// TIA Portal V15.1 export
// export: Created 2026-01-09T13:45:13.5597661Z, ExportSetting WithDefaults, WithReadOnly, DisplayName Totally Integrated Automation Portal, DisplayVersion V15.1 Update 8, DisplayName TIA Portal Openness, DisplayVersion V15.1 Update 8, DisplayName STEP 7 Professional, DisplayVersion V15.1 Update 8, DisplayName WinCC Advanced, DisplayVersion V15.1 Update 8
FUNCTION_BLOCK "11. LOGIC CAN"   // FB11, LAD
{ S7_Optimized_Access := 'TRUE' }
VERSION : 0.1
// stored: AutoNumber true, CodeModifiedDate 2025-08-27T17:14:05.4937984Z, CompileDate 2025-08-30T17:40:35.0335687Z, CreationDate 2024-10-12T12:36:08.0193576Z, DownloadWithoutReinit false, HandleErrorsWithinBlock false, InterfaceModifiedDate 2023-12-21T19:23:23.4270206Z, IsConsistent true, IsIECCheckEnabled false, IsKnowHowProtected false, IsRetainMemResEnabled false, IsWriteProtected false, LibraryConformanceStatus The object is library-conformant., MemoryReserve 100, ModifiedDate 2025-08-27T17:14:05.4937984Z, ParameterModified 2023-12-21T19:23:23.4270206Z, PLCSimAdvancedSupport false, SetENOAutomatically False, StructureModified 2023-12-21T19:23:23.4270206Z, UDAEnableTagReadback false
   VAR_INPUT
      LOGIC_1 : Real;
      LOGIC_2 : Real;
      LOGIC_3 : Real;
      "THC_1.1" : Bool;
      "THC_1.2" : Bool;
      "THC_2.1" : Bool;
      "THC_2.2" : Bool;
      "THC_3.1" : Bool;
      "THC_3.2" : Bool;
      "THC_4.1" : Bool;
      "THC_4.2" : Bool;
      "THC_5.1" : Bool;
      "THC_5.2" : Bool;
      "THC_6.1" : Bool;
      "THC_6.2" : Bool;
   END_VAR
   VAR_OUTPUT
      "OUT_LGOIC_1.1" : Bool;
      "OUT_LGOIC_1.2" : Bool;
      "OUT_LGOIC_2.1" : Bool;
      "OUT_LGOIC_2.2" : Bool;
      "OUT_LGOIC_3.1" : Bool;
      "OUT_LGOIC_3.2" : Bool;
      "OUT_LGOIC_4.1" : Bool;
      "OUT_LGOIC_4.2" : Bool;
      "OUT_LGOIC_5.1" : Bool;
      "OUT_LGOIC_5.2" : Bool;
      "OUT_LGOIC_6.1" : Bool;
      "OUT_LGOIC_6.2" : Bool;
   END_VAR
BEGIN

REGION Network 1: OUT1
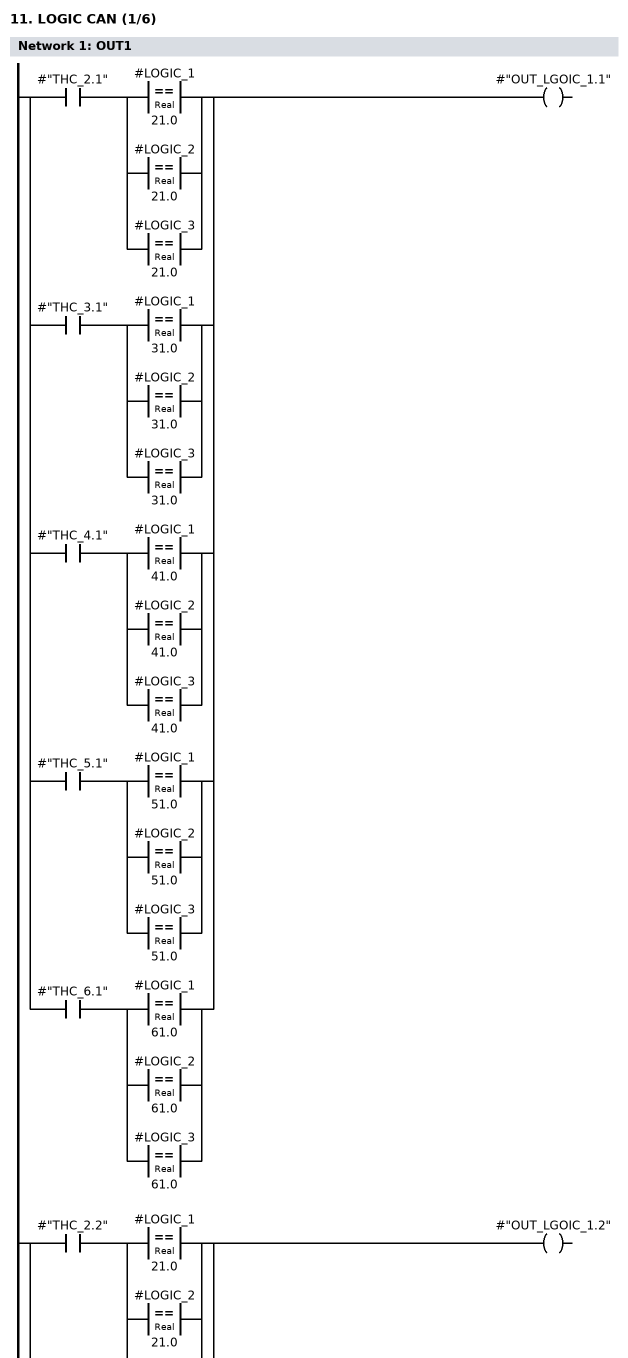
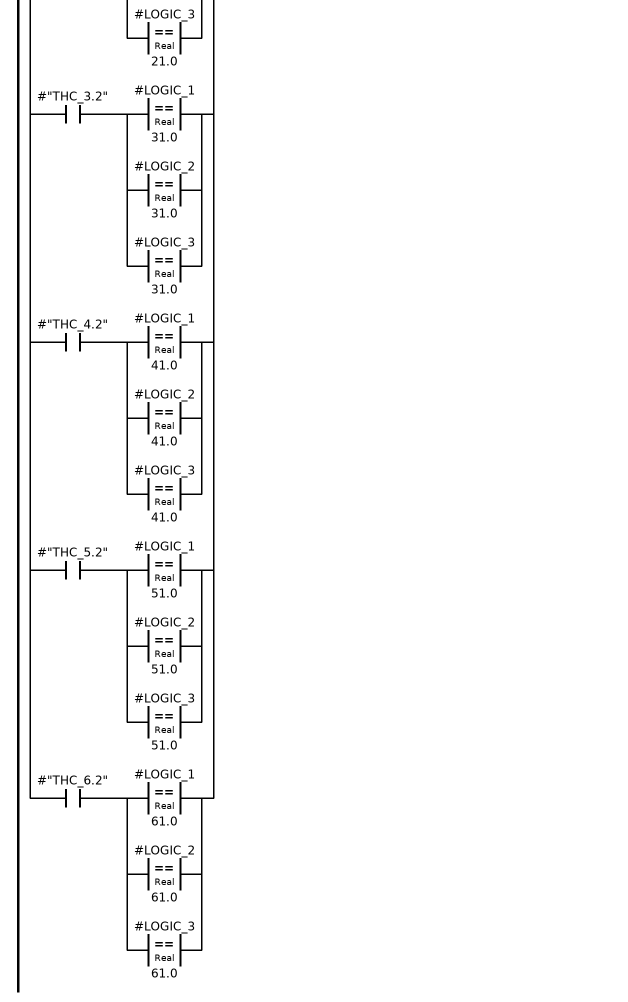
   RUNG wire#powerrail
      Contact( #"THC_2.1" )
      wire#w1
      { S7_Templates := "SrcType := Real" } EQ_Contact(in1 := #LOGIC_1, in2 := 21.0)
      wire#w2
      Coil( #"OUT_LGOIC_1.1" )
   END_RUNG
   RUNG wire#w1
      { S7_Templates := "SrcType := Real" } EQ_Contact(in1 := #LOGIC_2, in2 := 21.0)
   END_RUNG wire#w2
   RUNG wire#w1
      { S7_Templates := "SrcType := Real" } EQ_Contact(in1 := #LOGIC_3, in2 := 21.0)
   END_RUNG wire#w2
   RUNG wire#powerrail
      Contact( #"THC_3.1" )
      wire#w3
      { S7_Templates := "SrcType := Real" } EQ_Contact(in1 := #LOGIC_1, in2 := 31.0)
   END_RUNG wire#w2
   RUNG wire#w3
      { S7_Templates := "SrcType := Real" } EQ_Contact(in1 := #LOGIC_2, in2 := 31.0)
   END_RUNG wire#w2
   RUNG wire#w3
      { S7_Templates := "SrcType := Real" } EQ_Contact(in1 := #LOGIC_3, in2 := 31.0)
   END_RUNG wire#w2
   RUNG wire#powerrail
      Contact( #"THC_4.1" )
      wire#w4
      { S7_Templates := "SrcType := Real" } EQ_Contact(in1 := #LOGIC_1, in2 := 41.0)
   END_RUNG wire#w2
   RUNG wire#w4
      { S7_Templates := "SrcType := Real" } EQ_Contact(in1 := #LOGIC_2, in2 := 41.0)
   END_RUNG wire#w2
   RUNG wire#w4
      { S7_Templates := "SrcType := Real" } EQ_Contact(in1 := #LOGIC_3, in2 := 41.0)
   END_RUNG wire#w2
   RUNG wire#powerrail
      Contact( #"THC_5.1" )
      wire#w5
      { S7_Templates := "SrcType := Real" } EQ_Contact(in1 := #LOGIC_1, in2 := 51.0)
   END_RUNG wire#w2
   RUNG wire#w5
      { S7_Templates := "SrcType := Real" } EQ_Contact(in1 := #LOGIC_2, in2 := 51.0)
   END_RUNG wire#w2
   RUNG wire#w5
      { S7_Templates := "SrcType := Real" } EQ_Contact(in1 := #LOGIC_3, in2 := 51.0)
   END_RUNG wire#w2
   RUNG wire#powerrail
      Contact( #"THC_6.1" )
      wire#w6
      { S7_Templates := "SrcType := Real" } EQ_Contact(in1 := #LOGIC_1, in2 := 61.0)
   END_RUNG wire#w2
   RUNG wire#w6
      { S7_Templates := "SrcType := Real" } EQ_Contact(in1 := #LOGIC_2, in2 := 61.0)
   END_RUNG wire#w2
   RUNG wire#w6
      { S7_Templates := "SrcType := Real" } EQ_Contact(in1 := #LOGIC_3, in2 := 61.0)
   END_RUNG wire#w2
   RUNG wire#powerrail
      Contact( #"THC_2.2" )
      wire#w7
      { S7_Templates := "SrcType := Real" } EQ_Contact(in1 := #LOGIC_1, in2 := 21.0)
      wire#w8
      Coil( #"OUT_LGOIC_1.2" )
   END_RUNG
   RUNG wire#w7
      { S7_Templates := "SrcType := Real" } EQ_Contact(in1 := #LOGIC_2, in2 := 21.0)
   END_RUNG wire#w8
   RUNG wire#w7
      { S7_Templates := "SrcType := Real" } EQ_Contact(in1 := #LOGIC_3, in2 := 21.0)
   END_RUNG wire#w8
   RUNG wire#powerrail
      Contact( #"THC_3.2" )
      wire#w9
      { S7_Templates := "SrcType := Real" } EQ_Contact(in1 := #LOGIC_1, in2 := 31.0)
   END_RUNG wire#w8
   RUNG wire#w9
      { S7_Templates := "SrcType := Real" } EQ_Contact(in1 := #LOGIC_2, in2 := 31.0)
   END_RUNG wire#w8
   RUNG wire#w9
      { S7_Templates := "SrcType := Real" } EQ_Contact(in1 := #LOGIC_3, in2 := 31.0)
   END_RUNG wire#w8
   RUNG wire#powerrail
      Contact( #"THC_4.2" )
      wire#w10
      { S7_Templates := "SrcType := Real" } EQ_Contact(in1 := #LOGIC_1, in2 := 41.0)
   END_RUNG wire#w8
   RUNG wire#w10
      { S7_Templates := "SrcType := Real" } EQ_Contact(in1 := #LOGIC_2, in2 := 41.0)
   END_RUNG wire#w8
   RUNG wire#w10
      { S7_Templates := "SrcType := Real" } EQ_Contact(in1 := #LOGIC_3, in2 := 41.0)
   END_RUNG wire#w8
   RUNG wire#powerrail
      Contact( #"THC_5.2" )
      wire#w11
      { S7_Templates := "SrcType := Real" } EQ_Contact(in1 := #LOGIC_1, in2 := 51.0)
   END_RUNG wire#w8
   RUNG wire#w11
      { S7_Templates := "SrcType := Real" } EQ_Contact(in1 := #LOGIC_2, in2 := 51.0)
   END_RUNG wire#w8
   RUNG wire#w11
      { S7_Templates := "SrcType := Real" } EQ_Contact(in1 := #LOGIC_3, in2 := 51.0)
   END_RUNG wire#w8
   RUNG wire#powerrail
      Contact( #"THC_6.2" )
      wire#w12
      { S7_Templates := "SrcType := Real" } EQ_Contact(in1 := #LOGIC_1, in2 := 61.0)
   END_RUNG wire#w8
   RUNG wire#w12
      { S7_Templates := "SrcType := Real" } EQ_Contact(in1 := #LOGIC_2, in2 := 61.0)
   END_RUNG wire#w8
   RUNG wire#w12
      { S7_Templates := "SrcType := Real" } EQ_Contact(in1 := #LOGIC_3, in2 := 61.0)
   END_RUNG wire#w8
   // the same network as SCL:
   #"OUT_LGOIC_1.1" := (#"THC_2.1" AND ((#LOGIC_1 = 21.0) OR (#LOGIC_2 = 21.0) OR (#LOGIC_3 = 21.0))) OR (#"THC_3.1" AND ((#LOGIC_1 = 31.0) OR (#LOGIC_2 = 31.0) OR (#LOGIC_3 = 31.0))) OR (#"THC_4.1" AND ((#LOGIC_1 = 41.0) OR (#LOGIC_2 = 41.0) OR (#LOGIC_3 = 41.0))) OR (#"THC_5.1" AND ((#LOGIC_1 = 51.0) OR (#LOGIC_2 = 51.0) OR (#LOGIC_3 = 51.0))) OR (#"THC_6.1" AND ((#LOGIC_1 = 61.0) OR (#LOGIC_2 = 61.0) OR (#LOGIC_3 = 61.0)));
   #"OUT_LGOIC_1.2" := (#"THC_2.2" AND ((#LOGIC_1 = 21.0) OR (#LOGIC_2 = 21.0) OR (#LOGIC_3 = 21.0))) OR (#"THC_3.2" AND ((#LOGIC_1 = 31.0) OR (#LOGIC_2 = 31.0) OR (#LOGIC_3 = 31.0))) OR (#"THC_4.2" AND ((#LOGIC_1 = 41.0) OR (#LOGIC_2 = 41.0) OR (#LOGIC_3 = 41.0))) OR (#"THC_5.2" AND ((#LOGIC_1 = 51.0) OR (#LOGIC_2 = 51.0) OR (#LOGIC_3 = 51.0))) OR (#"THC_6.2" AND ((#LOGIC_1 = 61.0) OR (#LOGIC_2 = 61.0) OR (#LOGIC_3 = 61.0)));
END_REGION

REGION Network 2: OUT2
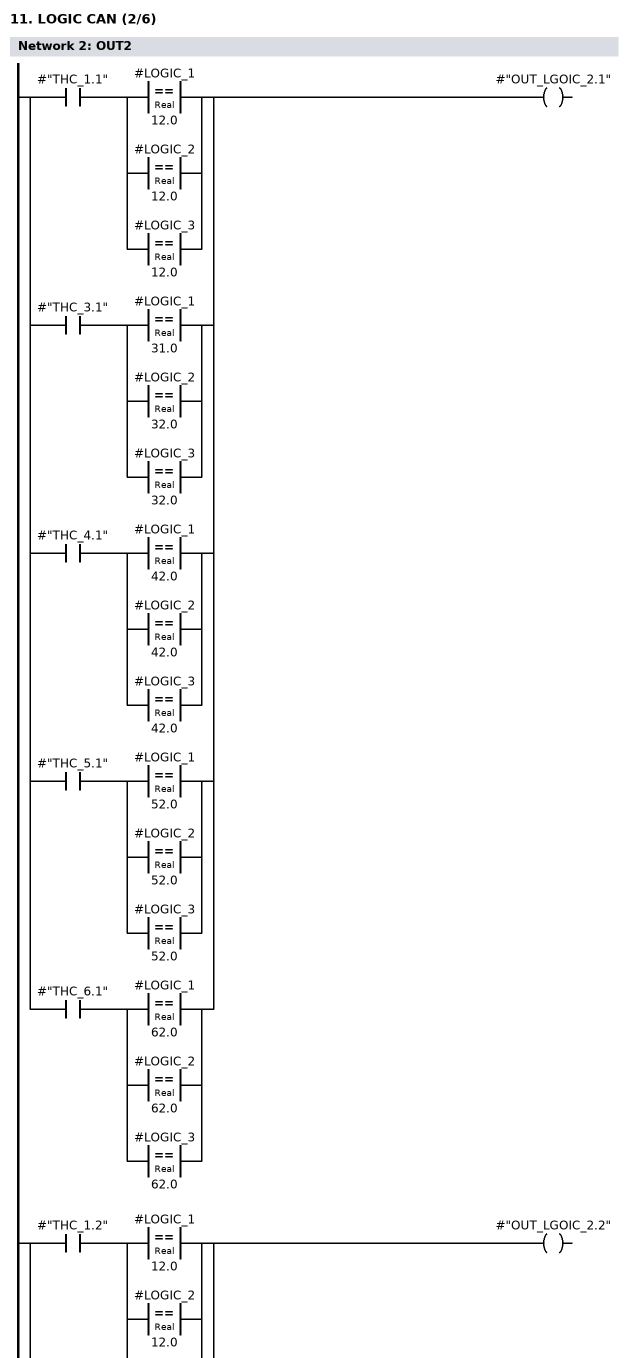
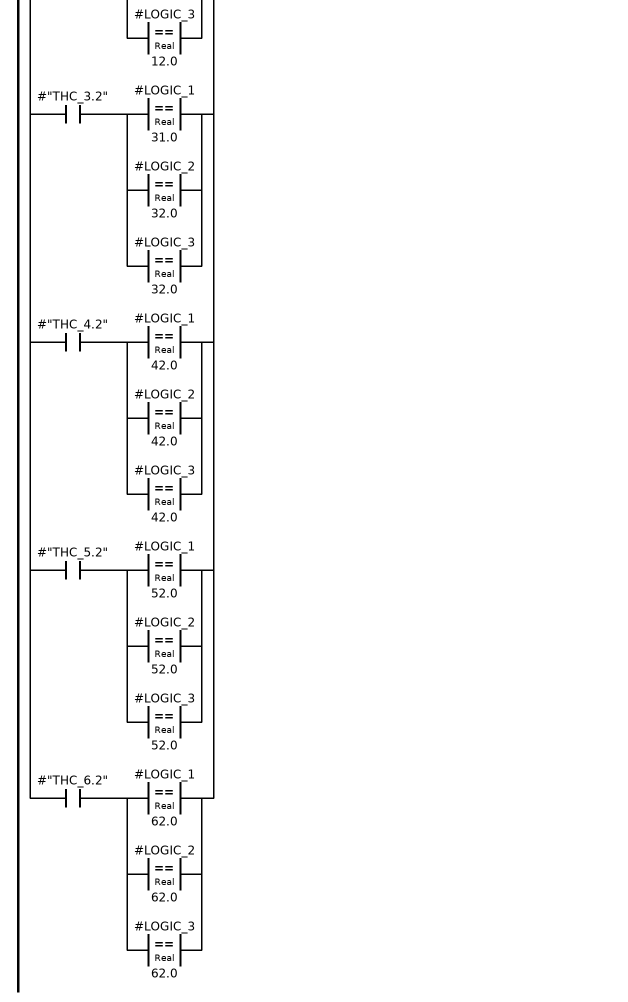
   RUNG wire#powerrail
      Contact( #"THC_1.1" )
      wire#w1
      { S7_Templates := "SrcType := Real" } EQ_Contact(in1 := #LOGIC_1, in2 := 12.0)
      wire#w2
      Coil( #"OUT_LGOIC_2.1" )
   END_RUNG
   RUNG wire#w1
      { S7_Templates := "SrcType := Real" } EQ_Contact(in1 := #LOGIC_2, in2 := 12.0)
   END_RUNG wire#w2
   RUNG wire#w1
      { S7_Templates := "SrcType := Real" } EQ_Contact(in1 := #LOGIC_3, in2 := 12.0)
   END_RUNG wire#w2
   RUNG wire#powerrail
      Contact( #"THC_3.1" )
      wire#w3
      { S7_Templates := "SrcType := Real" } EQ_Contact(in1 := #LOGIC_1, in2 := 31.0)
   END_RUNG wire#w2
   RUNG wire#w3
      { S7_Templates := "SrcType := Real" } EQ_Contact(in1 := #LOGIC_2, in2 := 32.0)
   END_RUNG wire#w2
   RUNG wire#w3
      { S7_Templates := "SrcType := Real" } EQ_Contact(in1 := #LOGIC_3, in2 := 32.0)
   END_RUNG wire#w2
   RUNG wire#powerrail
      Contact( #"THC_4.1" )
      wire#w4
      { S7_Templates := "SrcType := Real" } EQ_Contact(in1 := #LOGIC_1, in2 := 42.0)
   END_RUNG wire#w2
   RUNG wire#w4
      { S7_Templates := "SrcType := Real" } EQ_Contact(in1 := #LOGIC_2, in2 := 42.0)
   END_RUNG wire#w2
   RUNG wire#w4
      { S7_Templates := "SrcType := Real" } EQ_Contact(in1 := #LOGIC_3, in2 := 42.0)
   END_RUNG wire#w2
   RUNG wire#powerrail
      Contact( #"THC_5.1" )
      wire#w5
      { S7_Templates := "SrcType := Real" } EQ_Contact(in1 := #LOGIC_1, in2 := 52.0)
   END_RUNG wire#w2
   RUNG wire#w5
      { S7_Templates := "SrcType := Real" } EQ_Contact(in1 := #LOGIC_2, in2 := 52.0)
   END_RUNG wire#w2
   RUNG wire#w5
      { S7_Templates := "SrcType := Real" } EQ_Contact(in1 := #LOGIC_3, in2 := 52.0)
   END_RUNG wire#w2
   RUNG wire#powerrail
      Contact( #"THC_6.1" )
      wire#w6
      { S7_Templates := "SrcType := Real" } EQ_Contact(in1 := #LOGIC_1, in2 := 62.0)
   END_RUNG wire#w2
   RUNG wire#w6
      { S7_Templates := "SrcType := Real" } EQ_Contact(in1 := #LOGIC_2, in2 := 62.0)
   END_RUNG wire#w2
   RUNG wire#w6
      { S7_Templates := "SrcType := Real" } EQ_Contact(in1 := #LOGIC_3, in2 := 62.0)
   END_RUNG wire#w2
   RUNG wire#powerrail
      Contact( #"THC_1.2" )
      wire#w7
      { S7_Templates := "SrcType := Real" } EQ_Contact(in1 := #LOGIC_1, in2 := 12.0)
      wire#w8
      Coil( #"OUT_LGOIC_2.2" )
   END_RUNG
   RUNG wire#w7
      { S7_Templates := "SrcType := Real" } EQ_Contact(in1 := #LOGIC_2, in2 := 12.0)
   END_RUNG wire#w8
   RUNG wire#w7
      { S7_Templates := "SrcType := Real" } EQ_Contact(in1 := #LOGIC_3, in2 := 12.0)
   END_RUNG wire#w8
   RUNG wire#powerrail
      Contact( #"THC_3.2" )
      wire#w9
      { S7_Templates := "SrcType := Real" } EQ_Contact(in1 := #LOGIC_1, in2 := 31.0)
   END_RUNG wire#w8
   RUNG wire#w9
      { S7_Templates := "SrcType := Real" } EQ_Contact(in1 := #LOGIC_2, in2 := 32.0)
   END_RUNG wire#w8
   RUNG wire#w9
      { S7_Templates := "SrcType := Real" } EQ_Contact(in1 := #LOGIC_3, in2 := 32.0)
   END_RUNG wire#w8
   RUNG wire#powerrail
      Contact( #"THC_4.2" )
      wire#w10
      { S7_Templates := "SrcType := Real" } EQ_Contact(in1 := #LOGIC_1, in2 := 42.0)
   END_RUNG wire#w8
   RUNG wire#w10
      { S7_Templates := "SrcType := Real" } EQ_Contact(in1 := #LOGIC_2, in2 := 42.0)
   END_RUNG wire#w8
   RUNG wire#w10
      { S7_Templates := "SrcType := Real" } EQ_Contact(in1 := #LOGIC_3, in2 := 42.0)
   END_RUNG wire#w8
   RUNG wire#powerrail
      Contact( #"THC_5.2" )
      wire#w11
      { S7_Templates := "SrcType := Real" } EQ_Contact(in1 := #LOGIC_1, in2 := 52.0)
   END_RUNG wire#w8
   RUNG wire#w11
      { S7_Templates := "SrcType := Real" } EQ_Contact(in1 := #LOGIC_2, in2 := 52.0)
   END_RUNG wire#w8
   RUNG wire#w11
      { S7_Templates := "SrcType := Real" } EQ_Contact(in1 := #LOGIC_3, in2 := 52.0)
   END_RUNG wire#w8
   RUNG wire#powerrail
      Contact( #"THC_6.2" )
      wire#w12
      { S7_Templates := "SrcType := Real" } EQ_Contact(in1 := #LOGIC_1, in2 := 62.0)
   END_RUNG wire#w8
   RUNG wire#w12
      { S7_Templates := "SrcType := Real" } EQ_Contact(in1 := #LOGIC_2, in2 := 62.0)
   END_RUNG wire#w8
   RUNG wire#w12
      { S7_Templates := "SrcType := Real" } EQ_Contact(in1 := #LOGIC_3, in2 := 62.0)
   END_RUNG wire#w8
   // the same network as SCL:
   #"OUT_LGOIC_2.1" := (#"THC_1.1" AND ((#LOGIC_1 = 12.0) OR (#LOGIC_2 = 12.0) OR (#LOGIC_3 = 12.0))) OR (#"THC_3.1" AND ((#LOGIC_1 = 31.0) OR (#LOGIC_2 = 32.0) OR (#LOGIC_3 = 32.0))) OR (#"THC_4.1" AND ((#LOGIC_1 = 42.0) OR (#LOGIC_2 = 42.0) OR (#LOGIC_3 = 42.0))) OR (#"THC_5.1" AND ((#LOGIC_1 = 52.0) OR (#LOGIC_2 = 52.0) OR (#LOGIC_3 = 52.0))) OR (#"THC_6.1" AND ((#LOGIC_1 = 62.0) OR (#LOGIC_2 = 62.0) OR (#LOGIC_3 = 62.0)));
   #"OUT_LGOIC_2.2" := (#"THC_1.2" AND ((#LOGIC_1 = 12.0) OR (#LOGIC_2 = 12.0) OR (#LOGIC_3 = 12.0))) OR (#"THC_3.2" AND ((#LOGIC_1 = 31.0) OR (#LOGIC_2 = 32.0) OR (#LOGIC_3 = 32.0))) OR (#"THC_4.2" AND ((#LOGIC_1 = 42.0) OR (#LOGIC_2 = 42.0) OR (#LOGIC_3 = 42.0))) OR (#"THC_5.2" AND ((#LOGIC_1 = 52.0) OR (#LOGIC_2 = 52.0) OR (#LOGIC_3 = 52.0))) OR (#"THC_6.2" AND ((#LOGIC_1 = 62.0) OR (#LOGIC_2 = 62.0) OR (#LOGIC_3 = 62.0)));
END_REGION

REGION Network 3: OUT3
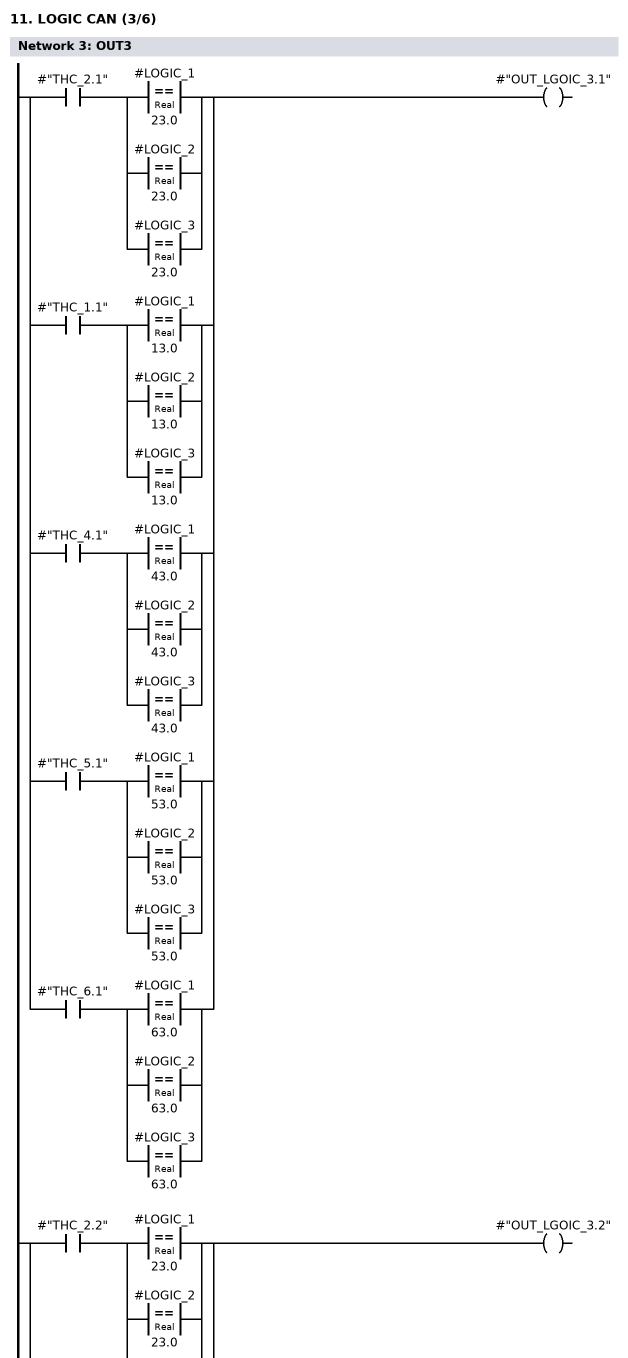
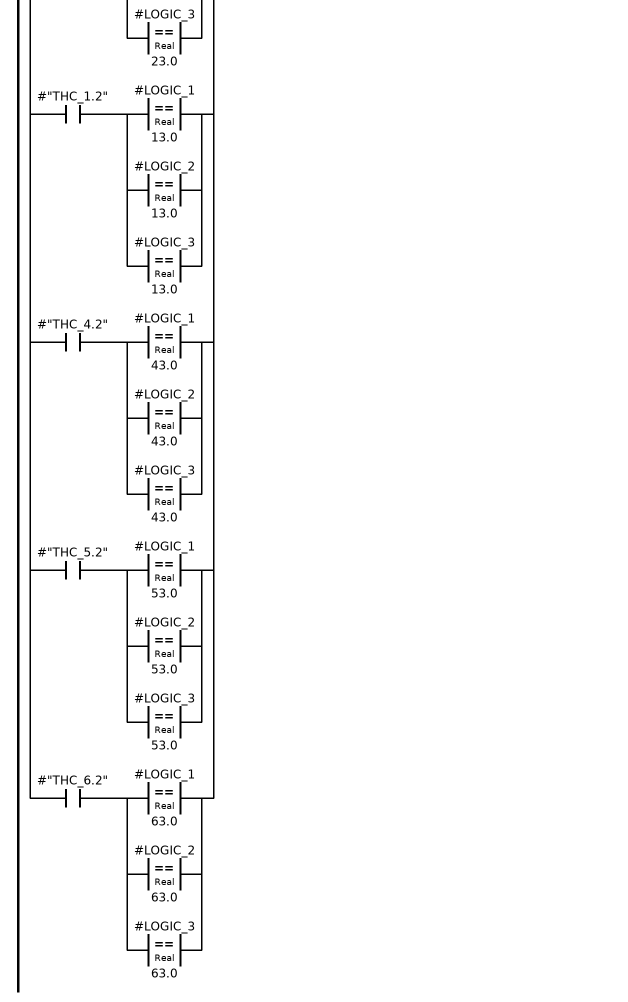
   RUNG wire#powerrail
      Contact( #"THC_2.1" )
      wire#w1
      { S7_Templates := "SrcType := Real" } EQ_Contact(in1 := #LOGIC_1, in2 := 23.0)
      wire#w2
      Coil( #"OUT_LGOIC_3.1" )
   END_RUNG
   RUNG wire#w1
      { S7_Templates := "SrcType := Real" } EQ_Contact(in1 := #LOGIC_2, in2 := 23.0)
   END_RUNG wire#w2
   RUNG wire#w1
      { S7_Templates := "SrcType := Real" } EQ_Contact(in1 := #LOGIC_3, in2 := 23.0)
   END_RUNG wire#w2
   RUNG wire#powerrail
      Contact( #"THC_1.1" )
      wire#w3
      { S7_Templates := "SrcType := Real" } EQ_Contact(in1 := #LOGIC_1, in2 := 13.0)
   END_RUNG wire#w2
   RUNG wire#w3
      { S7_Templates := "SrcType := Real" } EQ_Contact(in1 := #LOGIC_2, in2 := 13.0)
   END_RUNG wire#w2
   RUNG wire#w3
      { S7_Templates := "SrcType := Real" } EQ_Contact(in1 := #LOGIC_3, in2 := 13.0)
   END_RUNG wire#w2
   RUNG wire#powerrail
      Contact( #"THC_4.1" )
      wire#w4
      { S7_Templates := "SrcType := Real" } EQ_Contact(in1 := #LOGIC_1, in2 := 43.0)
   END_RUNG wire#w2
   RUNG wire#w4
      { S7_Templates := "SrcType := Real" } EQ_Contact(in1 := #LOGIC_2, in2 := 43.0)
   END_RUNG wire#w2
   RUNG wire#w4
      { S7_Templates := "SrcType := Real" } EQ_Contact(in1 := #LOGIC_3, in2 := 43.0)
   END_RUNG wire#w2
   RUNG wire#powerrail
      Contact( #"THC_5.1" )
      wire#w5
      { S7_Templates := "SrcType := Real" } EQ_Contact(in1 := #LOGIC_1, in2 := 53.0)
   END_RUNG wire#w2
   RUNG wire#w5
      { S7_Templates := "SrcType := Real" } EQ_Contact(in1 := #LOGIC_2, in2 := 53.0)
   END_RUNG wire#w2
   RUNG wire#w5
      { S7_Templates := "SrcType := Real" } EQ_Contact(in1 := #LOGIC_3, in2 := 53.0)
   END_RUNG wire#w2
   RUNG wire#powerrail
      Contact( #"THC_6.1" )
      wire#w6
      { S7_Templates := "SrcType := Real" } EQ_Contact(in1 := #LOGIC_1, in2 := 63.0)
   END_RUNG wire#w2
   RUNG wire#w6
      { S7_Templates := "SrcType := Real" } EQ_Contact(in1 := #LOGIC_2, in2 := 63.0)
   END_RUNG wire#w2
   RUNG wire#w6
      { S7_Templates := "SrcType := Real" } EQ_Contact(in1 := #LOGIC_3, in2 := 63.0)
   END_RUNG wire#w2
   RUNG wire#powerrail
      Contact( #"THC_2.2" )
      wire#w7
      { S7_Templates := "SrcType := Real" } EQ_Contact(in1 := #LOGIC_1, in2 := 23.0)
      wire#w8
      Coil( #"OUT_LGOIC_3.2" )
   END_RUNG
   RUNG wire#w7
      { S7_Templates := "SrcType := Real" } EQ_Contact(in1 := #LOGIC_2, in2 := 23.0)
   END_RUNG wire#w8
   RUNG wire#w7
      { S7_Templates := "SrcType := Real" } EQ_Contact(in1 := #LOGIC_3, in2 := 23.0)
   END_RUNG wire#w8
   RUNG wire#powerrail
      Contact( #"THC_1.2" )
      wire#w9
      { S7_Templates := "SrcType := Real" } EQ_Contact(in1 := #LOGIC_1, in2 := 13.0)
   END_RUNG wire#w8
   RUNG wire#w9
      { S7_Templates := "SrcType := Real" } EQ_Contact(in1 := #LOGIC_2, in2 := 13.0)
   END_RUNG wire#w8
   RUNG wire#w9
      { S7_Templates := "SrcType := Real" } EQ_Contact(in1 := #LOGIC_3, in2 := 13.0)
   END_RUNG wire#w8
   RUNG wire#powerrail
      Contact( #"THC_4.2" )
      wire#w10
      { S7_Templates := "SrcType := Real" } EQ_Contact(in1 := #LOGIC_1, in2 := 43.0)
   END_RUNG wire#w8
   RUNG wire#w10
      { S7_Templates := "SrcType := Real" } EQ_Contact(in1 := #LOGIC_2, in2 := 43.0)
   END_RUNG wire#w8
   RUNG wire#w10
      { S7_Templates := "SrcType := Real" } EQ_Contact(in1 := #LOGIC_3, in2 := 43.0)
   END_RUNG wire#w8
   RUNG wire#powerrail
      Contact( #"THC_5.2" )
      wire#w11
      { S7_Templates := "SrcType := Real" } EQ_Contact(in1 := #LOGIC_1, in2 := 53.0)
   END_RUNG wire#w8
   RUNG wire#w11
      { S7_Templates := "SrcType := Real" } EQ_Contact(in1 := #LOGIC_2, in2 := 53.0)
   END_RUNG wire#w8
   RUNG wire#w11
      { S7_Templates := "SrcType := Real" } EQ_Contact(in1 := #LOGIC_3, in2 := 53.0)
   END_RUNG wire#w8
   RUNG wire#powerrail
      Contact( #"THC_6.2" )
      wire#w12
      { S7_Templates := "SrcType := Real" } EQ_Contact(in1 := #LOGIC_1, in2 := 63.0)
   END_RUNG wire#w8
   RUNG wire#w12
      { S7_Templates := "SrcType := Real" } EQ_Contact(in1 := #LOGIC_2, in2 := 63.0)
   END_RUNG wire#w8
   RUNG wire#w12
      { S7_Templates := "SrcType := Real" } EQ_Contact(in1 := #LOGIC_3, in2 := 63.0)
   END_RUNG wire#w8
   // the same network as SCL:
   #"OUT_LGOIC_3.1" := (#"THC_2.1" AND ((#LOGIC_1 = 23.0) OR (#LOGIC_2 = 23.0) OR (#LOGIC_3 = 23.0))) OR (#"THC_1.1" AND ((#LOGIC_1 = 13.0) OR (#LOGIC_2 = 13.0) OR (#LOGIC_3 = 13.0))) OR (#"THC_4.1" AND ((#LOGIC_1 = 43.0) OR (#LOGIC_2 = 43.0) OR (#LOGIC_3 = 43.0))) OR (#"THC_5.1" AND ((#LOGIC_1 = 53.0) OR (#LOGIC_2 = 53.0) OR (#LOGIC_3 = 53.0))) OR (#"THC_6.1" AND ((#LOGIC_1 = 63.0) OR (#LOGIC_2 = 63.0) OR (#LOGIC_3 = 63.0)));
   #"OUT_LGOIC_3.2" := (#"THC_2.2" AND ((#LOGIC_1 = 23.0) OR (#LOGIC_2 = 23.0) OR (#LOGIC_3 = 23.0))) OR (#"THC_1.2" AND ((#LOGIC_1 = 13.0) OR (#LOGIC_2 = 13.0) OR (#LOGIC_3 = 13.0))) OR (#"THC_4.2" AND ((#LOGIC_1 = 43.0) OR (#LOGIC_2 = 43.0) OR (#LOGIC_3 = 43.0))) OR (#"THC_5.2" AND ((#LOGIC_1 = 53.0) OR (#LOGIC_2 = 53.0) OR (#LOGIC_3 = 53.0))) OR (#"THC_6.2" AND ((#LOGIC_1 = 63.0) OR (#LOGIC_2 = 63.0) OR (#LOGIC_3 = 63.0)));
END_REGION

REGION Network 4: OUT4
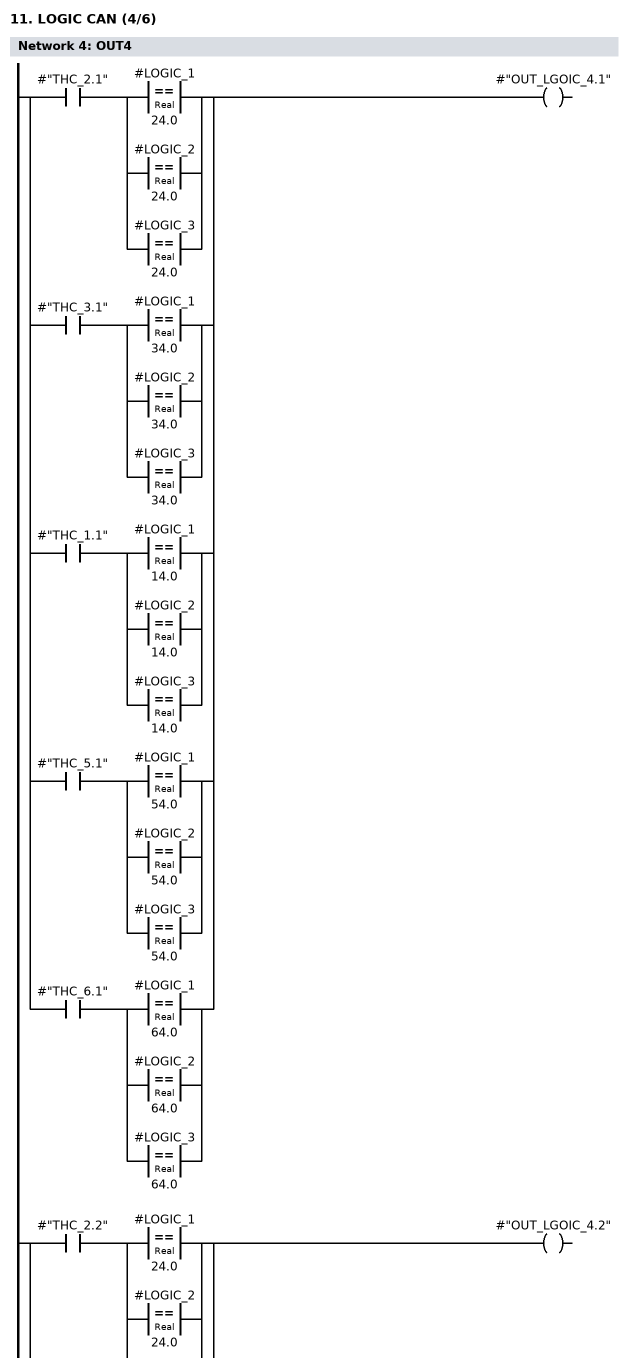
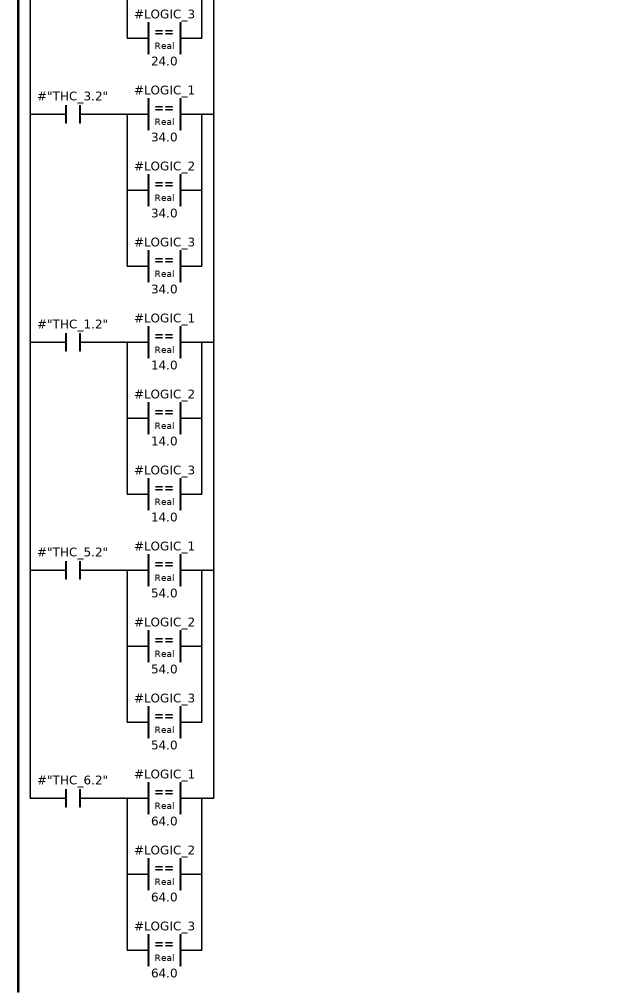
   RUNG wire#powerrail
      Contact( #"THC_2.1" )
      wire#w1
      { S7_Templates := "SrcType := Real" } EQ_Contact(in1 := #LOGIC_1, in2 := 24.0)
      wire#w2
      Coil( #"OUT_LGOIC_4.1" )
   END_RUNG
   RUNG wire#w1
      { S7_Templates := "SrcType := Real" } EQ_Contact(in1 := #LOGIC_2, in2 := 24.0)
   END_RUNG wire#w2
   RUNG wire#w1
      { S7_Templates := "SrcType := Real" } EQ_Contact(in1 := #LOGIC_3, in2 := 24.0)
   END_RUNG wire#w2
   RUNG wire#powerrail
      Contact( #"THC_3.1" )
      wire#w3
      { S7_Templates := "SrcType := Real" } EQ_Contact(in1 := #LOGIC_1, in2 := 34.0)
   END_RUNG wire#w2
   RUNG wire#w3
      { S7_Templates := "SrcType := Real" } EQ_Contact(in1 := #LOGIC_2, in2 := 34.0)
   END_RUNG wire#w2
   RUNG wire#w3
      { S7_Templates := "SrcType := Real" } EQ_Contact(in1 := #LOGIC_3, in2 := 34.0)
   END_RUNG wire#w2
   RUNG wire#powerrail
      Contact( #"THC_1.1" )
      wire#w4
      { S7_Templates := "SrcType := Real" } EQ_Contact(in1 := #LOGIC_1, in2 := 14.0)
   END_RUNG wire#w2
   RUNG wire#w4
      { S7_Templates := "SrcType := Real" } EQ_Contact(in1 := #LOGIC_2, in2 := 14.0)
   END_RUNG wire#w2
   RUNG wire#w4
      { S7_Templates := "SrcType := Real" } EQ_Contact(in1 := #LOGIC_3, in2 := 14.0)
   END_RUNG wire#w2
   RUNG wire#powerrail
      Contact( #"THC_5.1" )
      wire#w5
      { S7_Templates := "SrcType := Real" } EQ_Contact(in1 := #LOGIC_1, in2 := 54.0)
   END_RUNG wire#w2
   RUNG wire#w5
      { S7_Templates := "SrcType := Real" } EQ_Contact(in1 := #LOGIC_2, in2 := 54.0)
   END_RUNG wire#w2
   RUNG wire#w5
      { S7_Templates := "SrcType := Real" } EQ_Contact(in1 := #LOGIC_3, in2 := 54.0)
   END_RUNG wire#w2
   RUNG wire#powerrail
      Contact( #"THC_6.1" )
      wire#w6
      { S7_Templates := "SrcType := Real" } EQ_Contact(in1 := #LOGIC_1, in2 := 64.0)
   END_RUNG wire#w2
   RUNG wire#w6
      { S7_Templates := "SrcType := Real" } EQ_Contact(in1 := #LOGIC_2, in2 := 64.0)
   END_RUNG wire#w2
   RUNG wire#w6
      { S7_Templates := "SrcType := Real" } EQ_Contact(in1 := #LOGIC_3, in2 := 64.0)
   END_RUNG wire#w2
   RUNG wire#powerrail
      Contact( #"THC_2.2" )
      wire#w7
      { S7_Templates := "SrcType := Real" } EQ_Contact(in1 := #LOGIC_1, in2 := 24.0)
      wire#w8
      Coil( #"OUT_LGOIC_4.2" )
   END_RUNG
   RUNG wire#w7
      { S7_Templates := "SrcType := Real" } EQ_Contact(in1 := #LOGIC_2, in2 := 24.0)
   END_RUNG wire#w8
   RUNG wire#w7
      { S7_Templates := "SrcType := Real" } EQ_Contact(in1 := #LOGIC_3, in2 := 24.0)
   END_RUNG wire#w8
   RUNG wire#powerrail
      Contact( #"THC_3.2" )
      wire#w9
      { S7_Templates := "SrcType := Real" } EQ_Contact(in1 := #LOGIC_1, in2 := 34.0)
   END_RUNG wire#w8
   RUNG wire#w9
      { S7_Templates := "SrcType := Real" } EQ_Contact(in1 := #LOGIC_2, in2 := 34.0)
   END_RUNG wire#w8
   RUNG wire#w9
      { S7_Templates := "SrcType := Real" } EQ_Contact(in1 := #LOGIC_3, in2 := 34.0)
   END_RUNG wire#w8
   RUNG wire#powerrail
      Contact( #"THC_1.2" )
      wire#w10
      { S7_Templates := "SrcType := Real" } EQ_Contact(in1 := #LOGIC_1, in2 := 14.0)
   END_RUNG wire#w8
   RUNG wire#w10
      { S7_Templates := "SrcType := Real" } EQ_Contact(in1 := #LOGIC_2, in2 := 14.0)
   END_RUNG wire#w8
   RUNG wire#w10
      { S7_Templates := "SrcType := Real" } EQ_Contact(in1 := #LOGIC_3, in2 := 14.0)
   END_RUNG wire#w8
   RUNG wire#powerrail
      Contact( #"THC_5.2" )
      wire#w11
      { S7_Templates := "SrcType := Real" } EQ_Contact(in1 := #LOGIC_1, in2 := 54.0)
   END_RUNG wire#w8
   RUNG wire#w11
      { S7_Templates := "SrcType := Real" } EQ_Contact(in1 := #LOGIC_2, in2 := 54.0)
   END_RUNG wire#w8
   RUNG wire#w11
      { S7_Templates := "SrcType := Real" } EQ_Contact(in1 := #LOGIC_3, in2 := 54.0)
   END_RUNG wire#w8
   RUNG wire#powerrail
      Contact( #"THC_6.2" )
      wire#w12
      { S7_Templates := "SrcType := Real" } EQ_Contact(in1 := #LOGIC_1, in2 := 64.0)
   END_RUNG wire#w8
   RUNG wire#w12
      { S7_Templates := "SrcType := Real" } EQ_Contact(in1 := #LOGIC_2, in2 := 64.0)
   END_RUNG wire#w8
   RUNG wire#w12
      { S7_Templates := "SrcType := Real" } EQ_Contact(in1 := #LOGIC_3, in2 := 64.0)
   END_RUNG wire#w8
   // the same network as SCL:
   #"OUT_LGOIC_4.1" := (#"THC_2.1" AND ((#LOGIC_1 = 24.0) OR (#LOGIC_2 = 24.0) OR (#LOGIC_3 = 24.0))) OR (#"THC_3.1" AND ((#LOGIC_1 = 34.0) OR (#LOGIC_2 = 34.0) OR (#LOGIC_3 = 34.0))) OR (#"THC_1.1" AND ((#LOGIC_1 = 14.0) OR (#LOGIC_2 = 14.0) OR (#LOGIC_3 = 14.0))) OR (#"THC_5.1" AND ((#LOGIC_1 = 54.0) OR (#LOGIC_2 = 54.0) OR (#LOGIC_3 = 54.0))) OR (#"THC_6.1" AND ((#LOGIC_1 = 64.0) OR (#LOGIC_2 = 64.0) OR (#LOGIC_3 = 64.0)));
   #"OUT_LGOIC_4.2" := (#"THC_2.2" AND ((#LOGIC_1 = 24.0) OR (#LOGIC_2 = 24.0) OR (#LOGIC_3 = 24.0))) OR (#"THC_3.2" AND ((#LOGIC_1 = 34.0) OR (#LOGIC_2 = 34.0) OR (#LOGIC_3 = 34.0))) OR (#"THC_1.2" AND ((#LOGIC_1 = 14.0) OR (#LOGIC_2 = 14.0) OR (#LOGIC_3 = 14.0))) OR (#"THC_5.2" AND ((#LOGIC_1 = 54.0) OR (#LOGIC_2 = 54.0) OR (#LOGIC_3 = 54.0))) OR (#"THC_6.2" AND ((#LOGIC_1 = 64.0) OR (#LOGIC_2 = 64.0) OR (#LOGIC_3 = 64.0)));
END_REGION

REGION Network 5: OUT5
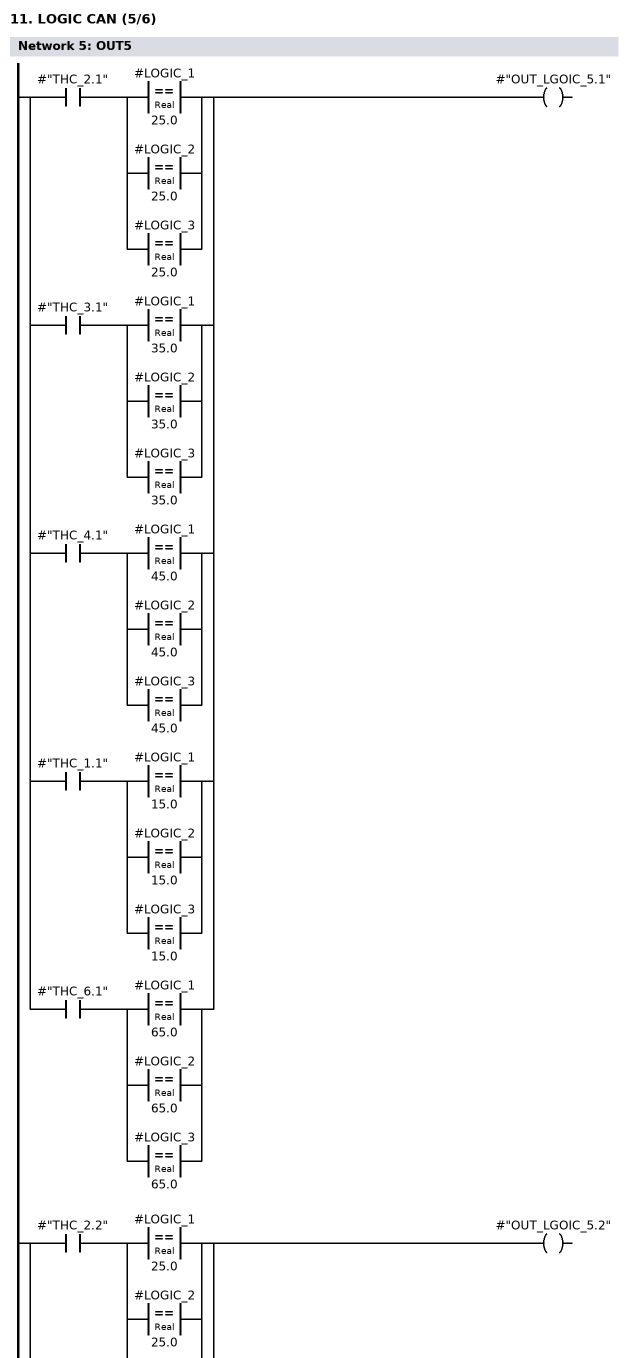
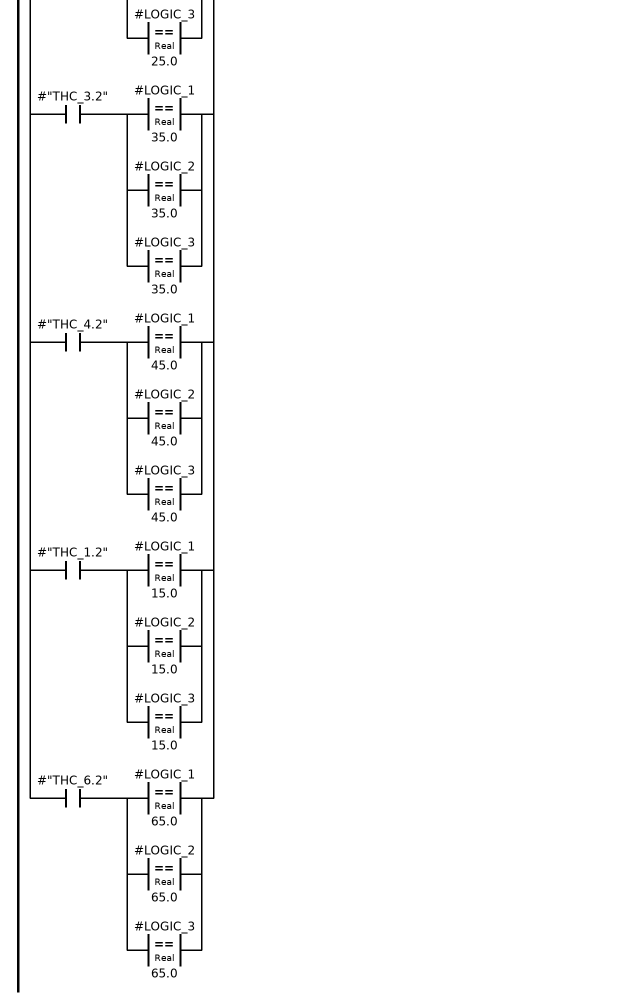
   RUNG wire#powerrail
      Contact( #"THC_2.1" )
      wire#w1
      { S7_Templates := "SrcType := Real" } EQ_Contact(in1 := #LOGIC_1, in2 := 25.0)
      wire#w2
      Coil( #"OUT_LGOIC_5.1" )
   END_RUNG
   RUNG wire#w1
      { S7_Templates := "SrcType := Real" } EQ_Contact(in1 := #LOGIC_2, in2 := 25.0)
   END_RUNG wire#w2
   RUNG wire#w1
      { S7_Templates := "SrcType := Real" } EQ_Contact(in1 := #LOGIC_3, in2 := 25.0)
   END_RUNG wire#w2
   RUNG wire#powerrail
      Contact( #"THC_3.1" )
      wire#w3
      { S7_Templates := "SrcType := Real" } EQ_Contact(in1 := #LOGIC_1, in2 := 35.0)
   END_RUNG wire#w2
   RUNG wire#w3
      { S7_Templates := "SrcType := Real" } EQ_Contact(in1 := #LOGIC_2, in2 := 35.0)
   END_RUNG wire#w2
   RUNG wire#w3
      { S7_Templates := "SrcType := Real" } EQ_Contact(in1 := #LOGIC_3, in2 := 35.0)
   END_RUNG wire#w2
   RUNG wire#powerrail
      Contact( #"THC_4.1" )
      wire#w4
      { S7_Templates := "SrcType := Real" } EQ_Contact(in1 := #LOGIC_1, in2 := 45.0)
   END_RUNG wire#w2
   RUNG wire#w4
      { S7_Templates := "SrcType := Real" } EQ_Contact(in1 := #LOGIC_2, in2 := 45.0)
   END_RUNG wire#w2
   RUNG wire#w4
      { S7_Templates := "SrcType := Real" } EQ_Contact(in1 := #LOGIC_3, in2 := 45.0)
   END_RUNG wire#w2
   RUNG wire#powerrail
      Contact( #"THC_1.1" )
      wire#w5
      { S7_Templates := "SrcType := Real" } EQ_Contact(in1 := #LOGIC_1, in2 := 15.0)
   END_RUNG wire#w2
   RUNG wire#w5
      { S7_Templates := "SrcType := Real" } EQ_Contact(in1 := #LOGIC_2, in2 := 15.0)
   END_RUNG wire#w2
   RUNG wire#w5
      { S7_Templates := "SrcType := Real" } EQ_Contact(in1 := #LOGIC_3, in2 := 15.0)
   END_RUNG wire#w2
   RUNG wire#powerrail
      Contact( #"THC_6.1" )
      wire#w6
      { S7_Templates := "SrcType := Real" } EQ_Contact(in1 := #LOGIC_1, in2 := 65.0)
   END_RUNG wire#w2
   RUNG wire#w6
      { S7_Templates := "SrcType := Real" } EQ_Contact(in1 := #LOGIC_2, in2 := 65.0)
   END_RUNG wire#w2
   RUNG wire#w6
      { S7_Templates := "SrcType := Real" } EQ_Contact(in1 := #LOGIC_3, in2 := 65.0)
   END_RUNG wire#w2
   RUNG wire#powerrail
      Contact( #"THC_2.2" )
      wire#w7
      { S7_Templates := "SrcType := Real" } EQ_Contact(in1 := #LOGIC_1, in2 := 25.0)
      wire#w8
      Coil( #"OUT_LGOIC_5.2" )
   END_RUNG
   RUNG wire#w7
      { S7_Templates := "SrcType := Real" } EQ_Contact(in1 := #LOGIC_2, in2 := 25.0)
   END_RUNG wire#w8
   RUNG wire#w7
      { S7_Templates := "SrcType := Real" } EQ_Contact(in1 := #LOGIC_3, in2 := 25.0)
   END_RUNG wire#w8
   RUNG wire#powerrail
      Contact( #"THC_3.2" )
      wire#w9
      { S7_Templates := "SrcType := Real" } EQ_Contact(in1 := #LOGIC_1, in2 := 35.0)
   END_RUNG wire#w8
   RUNG wire#w9
      { S7_Templates := "SrcType := Real" } EQ_Contact(in1 := #LOGIC_2, in2 := 35.0)
   END_RUNG wire#w8
   RUNG wire#w9
      { S7_Templates := "SrcType := Real" } EQ_Contact(in1 := #LOGIC_3, in2 := 35.0)
   END_RUNG wire#w8
   RUNG wire#powerrail
      Contact( #"THC_4.2" )
      wire#w10
      { S7_Templates := "SrcType := Real" } EQ_Contact(in1 := #LOGIC_1, in2 := 45.0)
   END_RUNG wire#w8
   RUNG wire#w10
      { S7_Templates := "SrcType := Real" } EQ_Contact(in1 := #LOGIC_2, in2 := 45.0)
   END_RUNG wire#w8
   RUNG wire#w10
      { S7_Templates := "SrcType := Real" } EQ_Contact(in1 := #LOGIC_3, in2 := 45.0)
   END_RUNG wire#w8
   RUNG wire#powerrail
      Contact( #"THC_1.2" )
      wire#w11
      { S7_Templates := "SrcType := Real" } EQ_Contact(in1 := #LOGIC_1, in2 := 15.0)
   END_RUNG wire#w8
   RUNG wire#w11
      { S7_Templates := "SrcType := Real" } EQ_Contact(in1 := #LOGIC_2, in2 := 15.0)
   END_RUNG wire#w8
   RUNG wire#w11
      { S7_Templates := "SrcType := Real" } EQ_Contact(in1 := #LOGIC_3, in2 := 15.0)
   END_RUNG wire#w8
   RUNG wire#powerrail
      Contact( #"THC_6.2" )
      wire#w12
      { S7_Templates := "SrcType := Real" } EQ_Contact(in1 := #LOGIC_1, in2 := 65.0)
   END_RUNG wire#w8
   RUNG wire#w12
      { S7_Templates := "SrcType := Real" } EQ_Contact(in1 := #LOGIC_2, in2 := 65.0)
   END_RUNG wire#w8
   RUNG wire#w12
      { S7_Templates := "SrcType := Real" } EQ_Contact(in1 := #LOGIC_3, in2 := 65.0)
   END_RUNG wire#w8
   // the same network as SCL:
   #"OUT_LGOIC_5.1" := (#"THC_2.1" AND ((#LOGIC_1 = 25.0) OR (#LOGIC_2 = 25.0) OR (#LOGIC_3 = 25.0))) OR (#"THC_3.1" AND ((#LOGIC_1 = 35.0) OR (#LOGIC_2 = 35.0) OR (#LOGIC_3 = 35.0))) OR (#"THC_4.1" AND ((#LOGIC_1 = 45.0) OR (#LOGIC_2 = 45.0) OR (#LOGIC_3 = 45.0))) OR (#"THC_1.1" AND ((#LOGIC_1 = 15.0) OR (#LOGIC_2 = 15.0) OR (#LOGIC_3 = 15.0))) OR (#"THC_6.1" AND ((#LOGIC_1 = 65.0) OR (#LOGIC_2 = 65.0) OR (#LOGIC_3 = 65.0)));
   #"OUT_LGOIC_5.2" := (#"THC_2.2" AND ((#LOGIC_1 = 25.0) OR (#LOGIC_2 = 25.0) OR (#LOGIC_3 = 25.0))) OR (#"THC_3.2" AND ((#LOGIC_1 = 35.0) OR (#LOGIC_2 = 35.0) OR (#LOGIC_3 = 35.0))) OR (#"THC_4.2" AND ((#LOGIC_1 = 45.0) OR (#LOGIC_2 = 45.0) OR (#LOGIC_3 = 45.0))) OR (#"THC_1.2" AND ((#LOGIC_1 = 15.0) OR (#LOGIC_2 = 15.0) OR (#LOGIC_3 = 15.0))) OR (#"THC_6.2" AND ((#LOGIC_1 = 65.0) OR (#LOGIC_2 = 65.0) OR (#LOGIC_3 = 65.0)));
END_REGION

REGION Network 6: OUT6
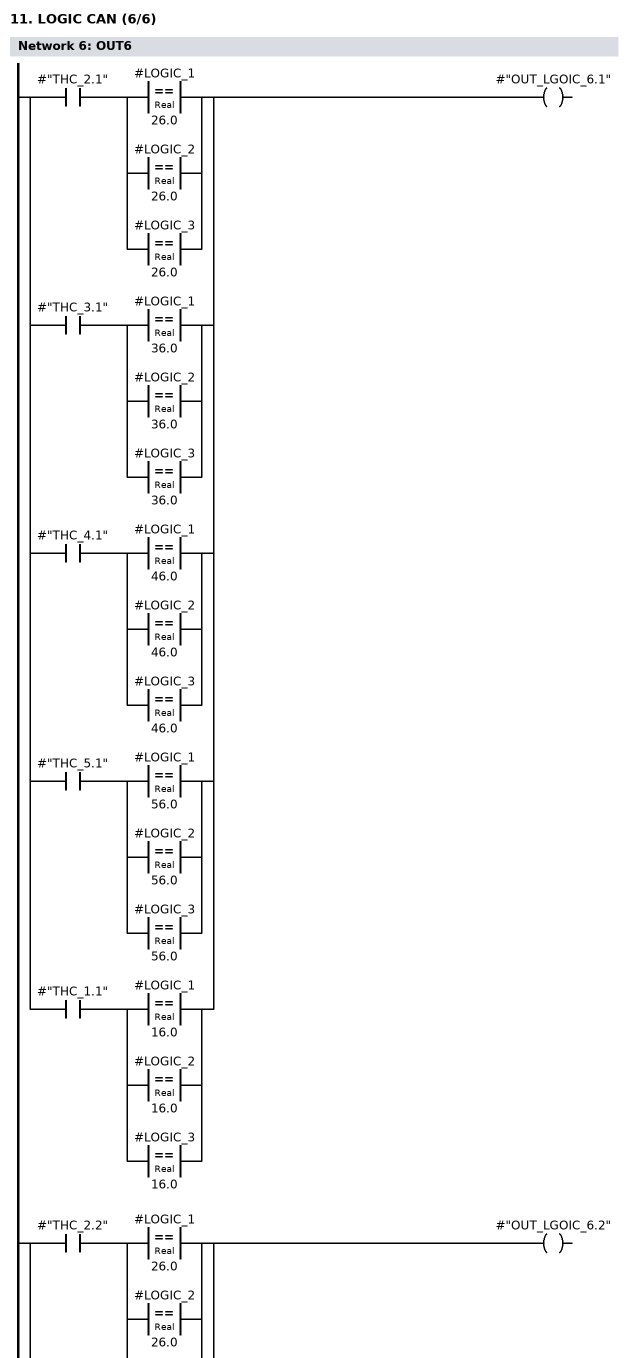
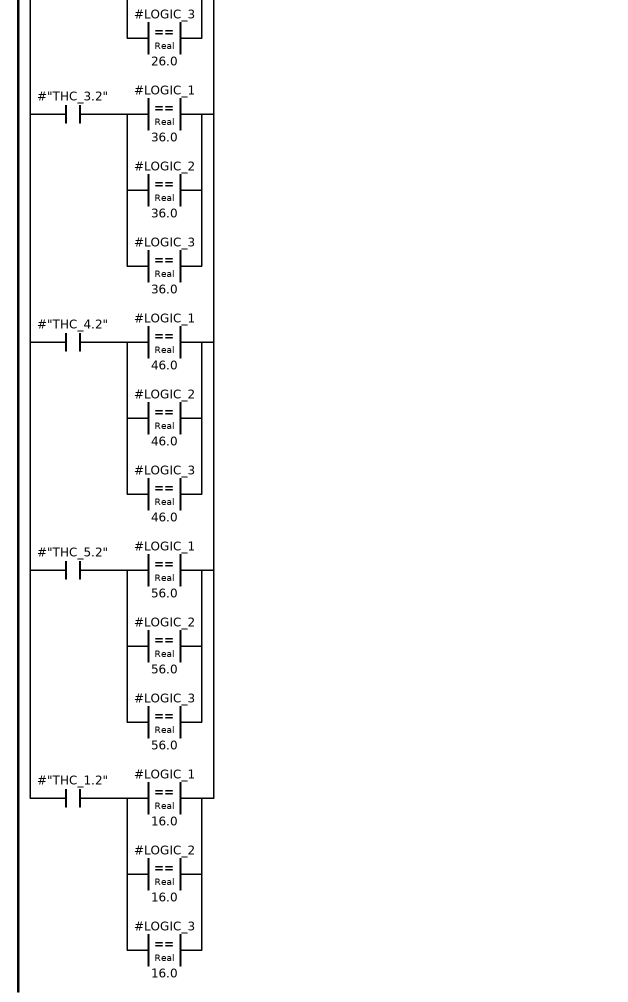
   RUNG wire#powerrail
      Contact( #"THC_2.1" )
      wire#w1
      { S7_Templates := "SrcType := Real" } EQ_Contact(in1 := #LOGIC_1, in2 := 26.0)
      wire#w2
      Coil( #"OUT_LGOIC_6.1" )
   END_RUNG
   RUNG wire#w1
      { S7_Templates := "SrcType := Real" } EQ_Contact(in1 := #LOGIC_2, in2 := 26.0)
   END_RUNG wire#w2
   RUNG wire#w1
      { S7_Templates := "SrcType := Real" } EQ_Contact(in1 := #LOGIC_3, in2 := 26.0)
   END_RUNG wire#w2
   RUNG wire#powerrail
      Contact( #"THC_3.1" )
      wire#w3
      { S7_Templates := "SrcType := Real" } EQ_Contact(in1 := #LOGIC_1, in2 := 36.0)
   END_RUNG wire#w2
   RUNG wire#w3
      { S7_Templates := "SrcType := Real" } EQ_Contact(in1 := #LOGIC_2, in2 := 36.0)
   END_RUNG wire#w2
   RUNG wire#w3
      { S7_Templates := "SrcType := Real" } EQ_Contact(in1 := #LOGIC_3, in2 := 36.0)
   END_RUNG wire#w2
   RUNG wire#powerrail
      Contact( #"THC_4.1" )
      wire#w4
      { S7_Templates := "SrcType := Real" } EQ_Contact(in1 := #LOGIC_1, in2 := 46.0)
   END_RUNG wire#w2
   RUNG wire#w4
      { S7_Templates := "SrcType := Real" } EQ_Contact(in1 := #LOGIC_2, in2 := 46.0)
   END_RUNG wire#w2
   RUNG wire#w4
      { S7_Templates := "SrcType := Real" } EQ_Contact(in1 := #LOGIC_3, in2 := 46.0)
   END_RUNG wire#w2
   RUNG wire#powerrail
      Contact( #"THC_5.1" )
      wire#w5
      { S7_Templates := "SrcType := Real" } EQ_Contact(in1 := #LOGIC_1, in2 := 56.0)
   END_RUNG wire#w2
   RUNG wire#w5
      { S7_Templates := "SrcType := Real" } EQ_Contact(in1 := #LOGIC_2, in2 := 56.0)
   END_RUNG wire#w2
   RUNG wire#w5
      { S7_Templates := "SrcType := Real" } EQ_Contact(in1 := #LOGIC_3, in2 := 56.0)
   END_RUNG wire#w2
   RUNG wire#powerrail
      Contact( #"THC_1.1" )
      wire#w6
      { S7_Templates := "SrcType := Real" } EQ_Contact(in1 := #LOGIC_1, in2 := 16.0)
   END_RUNG wire#w2
   RUNG wire#w6
      { S7_Templates := "SrcType := Real" } EQ_Contact(in1 := #LOGIC_2, in2 := 16.0)
   END_RUNG wire#w2
   RUNG wire#w6
      { S7_Templates := "SrcType := Real" } EQ_Contact(in1 := #LOGIC_3, in2 := 16.0)
   END_RUNG wire#w2
   RUNG wire#powerrail
      Contact( #"THC_2.2" )
      wire#w7
      { S7_Templates := "SrcType := Real" } EQ_Contact(in1 := #LOGIC_1, in2 := 26.0)
      wire#w8
      Coil( #"OUT_LGOIC_6.2" )
   END_RUNG
   RUNG wire#w7
      { S7_Templates := "SrcType := Real" } EQ_Contact(in1 := #LOGIC_2, in2 := 26.0)
   END_RUNG wire#w8
   RUNG wire#w7
      { S7_Templates := "SrcType := Real" } EQ_Contact(in1 := #LOGIC_3, in2 := 26.0)
   END_RUNG wire#w8
   RUNG wire#powerrail
      Contact( #"THC_3.2" )
      wire#w9
      { S7_Templates := "SrcType := Real" } EQ_Contact(in1 := #LOGIC_1, in2 := 36.0)
   END_RUNG wire#w8
   RUNG wire#w9
      { S7_Templates := "SrcType := Real" } EQ_Contact(in1 := #LOGIC_2, in2 := 36.0)
   END_RUNG wire#w8
   RUNG wire#w9
      { S7_Templates := "SrcType := Real" } EQ_Contact(in1 := #LOGIC_3, in2 := 36.0)
   END_RUNG wire#w8
   RUNG wire#powerrail
      Contact( #"THC_4.2" )
      wire#w10
      { S7_Templates := "SrcType := Real" } EQ_Contact(in1 := #LOGIC_1, in2 := 46.0)
   END_RUNG wire#w8
   RUNG wire#w10
      { S7_Templates := "SrcType := Real" } EQ_Contact(in1 := #LOGIC_2, in2 := 46.0)
   END_RUNG wire#w8
   RUNG wire#w10
      { S7_Templates := "SrcType := Real" } EQ_Contact(in1 := #LOGIC_3, in2 := 46.0)
   END_RUNG wire#w8
   RUNG wire#powerrail
      Contact( #"THC_5.2" )
      wire#w11
      { S7_Templates := "SrcType := Real" } EQ_Contact(in1 := #LOGIC_1, in2 := 56.0)
   END_RUNG wire#w8
   RUNG wire#w11
      { S7_Templates := "SrcType := Real" } EQ_Contact(in1 := #LOGIC_2, in2 := 56.0)
   END_RUNG wire#w8
   RUNG wire#w11
      { S7_Templates := "SrcType := Real" } EQ_Contact(in1 := #LOGIC_3, in2 := 56.0)
   END_RUNG wire#w8
   RUNG wire#powerrail
      Contact( #"THC_1.2" )
      wire#w12
      { S7_Templates := "SrcType := Real" } EQ_Contact(in1 := #LOGIC_1, in2 := 16.0)
   END_RUNG wire#w8
   RUNG wire#w12
      { S7_Templates := "SrcType := Real" } EQ_Contact(in1 := #LOGIC_2, in2 := 16.0)
   END_RUNG wire#w8
   RUNG wire#w12
      { S7_Templates := "SrcType := Real" } EQ_Contact(in1 := #LOGIC_3, in2 := 16.0)
   END_RUNG wire#w8
   // the same network as SCL:
   #"OUT_LGOIC_6.1" := (#"THC_2.1" AND ((#LOGIC_1 = 26.0) OR (#LOGIC_2 = 26.0) OR (#LOGIC_3 = 26.0))) OR (#"THC_3.1" AND ((#LOGIC_1 = 36.0) OR (#LOGIC_2 = 36.0) OR (#LOGIC_3 = 36.0))) OR (#"THC_4.1" AND ((#LOGIC_1 = 46.0) OR (#LOGIC_2 = 46.0) OR (#LOGIC_3 = 46.0))) OR (#"THC_5.1" AND ((#LOGIC_1 = 56.0) OR (#LOGIC_2 = 56.0) OR (#LOGIC_3 = 56.0))) OR (#"THC_1.1" AND ((#LOGIC_1 = 16.0) OR (#LOGIC_2 = 16.0) OR (#LOGIC_3 = 16.0)));
   #"OUT_LGOIC_6.2" := (#"THC_2.2" AND ((#LOGIC_1 = 26.0) OR (#LOGIC_2 = 26.0) OR (#LOGIC_3 = 26.0))) OR (#"THC_3.2" AND ((#LOGIC_1 = 36.0) OR (#LOGIC_2 = 36.0) OR (#LOGIC_3 = 36.0))) OR (#"THC_4.2" AND ((#LOGIC_1 = 46.0) OR (#LOGIC_2 = 46.0) OR (#LOGIC_3 = 46.0))) OR (#"THC_5.2" AND ((#LOGIC_1 = 56.0) OR (#LOGIC_2 = 56.0) OR (#LOGIC_3 = 56.0))) OR (#"THC_1.2" AND ((#LOGIC_1 = 16.0) OR (#LOGIC_2 = 16.0) OR (#LOGIC_3 = 16.0)));
END_REGION
END_FUNCTION_BLOCK
